KUKA KRL data list: AppFeedbackSPS.dat

&ACCESS RVP
&REL 1
&PARAM DISKPATH = TP/Tesla_Core
DEFDAT AppFeedbackSPS
; **************************************
; * Package:     TeslaCore             *
; * Release      V5.0.0                *
; * File:        AppFeedbackSPS.dat    *
; * Date:        04.2019               *
; * GUI Version: > = V8.3              *
; **************************************
;FOLD Application Feedback
;ENDFOLD (Application Feedback)
ENDDAT
